{attribute 'linkalways'} 
{attribute 'no_explicit_call' := 'This FB is a CLASS and must be accessed using methods or properties'}
{attribute 'enable_dynamic_creation'}
{attribute 'hide_all_locals'}
FUNCTION_BLOCK PUBLIC FINAL List EXTENDS Disposable IMPLEMENTS I_List
VAR
	memoryManager : FB_DynMem_Manager2;
	buffer : FB_DynMem_Buffer(ipMemMan := memoryManager);
	pArrayOfListNodes : POINTER TO I_ListNode;
	arrayCapacity : DINT;
	itemCount : DINT;
	eventEmitter : EventEmitter;
END_VAR

METHOD PUBLIC AddItem
VAR_INPUT
	Item : ANY;
END_VAR
VAR
	node : I_ListNode;
END_VAR
node := CreateNewNode(Item);
IF AddNodeLast(node) THEN
	EmitChangedEvent();
END_IF
END_METHOD

METHOD PRIVATE AddNodeAt : BOOL
VAR_INPUT
	Index : DINT;
	Node : I_ListNode;
END_VAR
VAR
	i : DINT;
END_VAR
IF Index = itemCount THEN
	IF AddNodeLast(Node) THEN
		AddNodeAt := TRUE;
	END_IF
	RETURN;
END_IF

IF Index > itemCount - 1 THEN
	RETURN;
END_IF

IF itemCount + 1 > arrayCapacity THEN
	IF NOT Grow() THEN
		RETURN;
	END_IF
END_IF

IF IsBufferPointerValid THEN
	//Move all excisting nodes up
	FOR i := itemCount - 1 TO Index BY -1 DO
		pArrayOfListNodes[i + 1] := pArrayOfListNodes[i];
		pArrayOfListNodes[i] := 0;
	END_FOR
	
	pArrayOfListNodes[Index] := Node;
	itemCount := itemCount + 1;
	
	AddNodeAt := TRUE;
END_IF
END_METHOD

METHOD PRIVATE AddNodeLast : BOOL
VAR_INPUT
	Node : I_ListNode;
END_VAR
IF itemCount = arrayCapacity THEN
    IF NOT Grow() THEN
		RETURN;
	END_IF
END_IF

IF IsBufferPointerValid THEN
	pArrayOfListNodes[itemCount] := Node;
	itemCount := itemCount + 1;
	
	AddNodeLast := TRUE;
END_IF
END_METHOD

PROPERTY PUBLIC Capacity : DINT
GET
Capacity := arrayCapacity;
END_GET
END_PROPERTY

METHOD Clear
VAR_INPUT
END_VAR
IF IsEmpty THEN
	RETURN;
END_IF

RemoveAllNodes();
EmitChangedEvent();
END_METHOD

METHOD Contains : BOOL
VAR_INPUT
	Item : ANY;
END_VAR
IF IsEmpty THEN
	RETURN;
END_IF

Contains := GetIndexOf(Item) > -1;
END_METHOD

PROPERTY PUBLIC Count : DINT
GET
Count := itemCount;
END_GET
END_PROPERTY

METHOD PRIVATE CreateNewNode : I_ListNode
VAR_INPUT
	Value : ANY;
END_VAR
VAR
	pNode : POINTER TO ListNode;
END_VAR
pNode := __NEW(ListNode(Source := Value));
CreateNewNode := pNode^;
END_METHOD

METHOD PRIVATE EmitChangedEvent
VAR
	pCollectionChangedEvent : POINTER TO CollectionChangedEvent;
END_VAR
pCollectionChangedEvent := __NEW(CollectionChangedEvent(Target := THIS^));
eventEmitter.Emit('OnChanged', pCollectionChangedEvent^);
pCollectionChangedEvent^.Dispose();
END_METHOD

METHOD PRIVATE EmitDisposedEvent
VAR
	pCollectionDisposedEvent : POINTER TO CollectionDisposedEvent;
END_VAR
pCollectionDisposedEvent := __NEW(CollectionDisposedEvent(Target := THIS^));
eventEmitter.Emit('OnDisposed', pCollectionDisposedEvent^);
pCollectionDisposedEvent^.Dispose();
END_METHOD

METHOD FB_exit : BOOL
VAR_INPUT
	bInCopyCode : BOOL; // if TRUE, the exit method is called for exiting an instance that is copied afterwards (online change).
END_VAR
VAR
END_VAR
IF bInCopyCode THEN
    RETURN;
END_IF

Clear();
buffer.DeleteBuffer();
EmitDisposedEvent();
END_METHOD

METHOD GetEnumerator : I_ForwardEnumerator
VAR
	pEnumerator : POINTER TO ListForwardEnumerator;
END_VAR
pEnumerator := __NEW(ListForwardEnumerator(Parent := THIS^));
GetEnumerator := pEnumerator^;
END_METHOD

METHOD PUBLIC GetIndexOf : DINT
VAR_INPUT
	Item : ANY;
END_VAR
VAR
	node : I_ListNode;
	i : DINT;
END_VAR
GetIndexOf := -1;

IF IsEmpty THEN
	RETURN;
END_IF

FOR i := 0 TO itemCount - 1 DO
	node := THIS^.Item(i);
	
	IF node.Equals(Item) THEN
		GetIndexOf := i;
		RETURN;
	END_IF
END_FOR
END_METHOD

METHOD PRIVATE Grow : BOOL
VAR
	node : I_ListNode;
END_VAR
VAR CONSTANT
	INITIAL_CAPACITY : DINT := 4;
END_VAR
IF arrayCapacity = 0 THEN
	arrayCapacity := INITIAL_CAPACITY;
ELSE
	arrayCapacity := arrayCapacity * 2;
END_IF

IF buffer.bAvailable THEN
	IF NOT buffer.Resize(nSize := DINT_TO_UDINT(arrayCapacity) * SIZEOF(node), bPreserve := TRUE, bReset := FALSE) THEN
		RETURN;
	END_IF
ELSE
	IF NOT buffer.CreateBuffer(nSize := DINT_TO_UDINT(arrayCapacity) * SIZEOF(node), bReset := TRUE) THEN
		RETURN;
	END_IF
END_IF

IF buffer.bAvailable THEN
	pArrayOfListNodes := buffer.pBuffer;
	
	IF IsBufferPointerValid THEN
		Grow := TRUE;
	END_IF
END_IF
END_METHOD

PROPERTY PRIVATE IsBufferPointerValid : BOOL
GET
IsBufferPointerValid := pArrayOfListNodes <> 0;
END_GET
END_PROPERTY

PROPERTY IsEmpty : BOOL
GET
IsEmpty := itemCount = 0;
END_GET
END_PROPERTY

METHOD PRIVATE IsNotValidIndex : BOOL
VAR_INPUT
	Index : DINT;
END_VAR
IsNotValidIndex := NOT IsValidIndex(Index);
END_METHOD

METHOD PRIVATE IsValidIndex : BOOL
VAR_INPUT
	Index : DINT;
END_VAR
IF Index < 0 THEN
	RETURN;
END_IF

IF Index >= itemCount THEN
	RETURN;
END_IF

IsValidIndex := TRUE;
END_METHOD

METHOD PRIVATE Item : I_ListNode
VAR_INPUT
	Index : DINT;
END_VAR
IF IsNotValidIndex(Index) THEN
	RETURN;
END_IF

IF IsBufferPointerValid THEN
	Item := pArrayOfListNodes[Index];
END_IF
END_METHOD

METHOD PUBLIC OffEvent
VAR_INPUT
	EventName : T_MaxString;
	EventHandler : I_EventHandler;
END_VAR
eventEmitter.OffEvent(EventName, EventHandler);
END_METHOD

METHOD PUBLIC OnceEvent
VAR_INPUT
	EventName : T_MaxString;
	EventHandler : I_EventHandler;
END_VAR
eventEmitter.OnceEvent(EventName, EventHandler);
END_METHOD

METHOD PUBLIC OnEvent
VAR_INPUT
	EventName : T_MaxString;
	EventHandler : I_EventHandler;
END_VAR
eventEmitter.OnEvent(EventName, EventHandler);
END_METHOD

METHOD PRIVATE RemoveAllNodes
VAR
	i : DINT;
END_VAR
FOR i := 0 TO itemCount - 1 DO
	IF pArrayOfListNodes[i] <> 0 THEN
		pArrayOfListNodes[i].Dispose();
	END_IF
END_FOR

itemCount := 0;
END_METHOD

METHOD PUBLIC TrimExcess
VAR
	node : I_ListNode;
END_VAR
IF arrayCapacity = 0 THEN
	RETURN;
END_IF

IF arrayCapacity = itemCount THEN
	RETURN;
END_IF

arrayCapacity := itemCount;
IF buffer.Resize(nSize := DINT_TO_UDINT(arrayCapacity) * SIZEOF(node), bPreserve := TRUE, bReset := FALSE) THEN
	pArrayOfListNodes := buffer.pBuffer;
ELSE
	pArrayOfListNodes := 0;
END_IF
END_METHOD

METHOD PUBLIC TryCopyTo : BOOL
VAR_INPUT
	Destination	: ANY;
END_VAR
TryCopyTo := TryCopyToLocation(Destination.pValue, DINT_TO_UDINT(Destination.diSize));
END_METHOD

METHOD PUBLIC TryCopyToLocation : BOOL
VAR_INPUT
	DestinationAddress : PVOID;
	DestinationSize : UDINT;
END_VAR
VAR
	i : DINT;
	requiredSize : UDINT;
	current : I_ListNode;
	pCurrent : PVOID;
END_VAR
IF IsEmpty THEN
    RETURN;
END_IF

//Compute required size
FOR i := 0 TO Count - 1 DO
    current := Item(i);
    requiredSize := requiredSize + current.DataSize;
END_FOR

//If destination size is to small abort
IF DestinationSize < requiredSize THEN
    RETURN;
END_IF

pCurrent := DestinationAddress;

FOR i := 0 TO Count - 1 DO
    current := Item(i);
    current.TryGetTo(pCurrent, current.DataSize);
    pCurrent := pCurrent + current.DataSize;
END_FOR
END_METHOD

METHOD PUBLIC TryGetByIndex : BOOL
VAR_INPUT
	Index : DINT;
	Destination : ANY;
END_VAR
VAR
	node : I_ListNode;
END_VAR
node := Item(Index);

IF node = 0 THEN
	RETURN;
END_IF

TryGetByIndex := node.TryGet(Destination);
END_METHOD

METHOD PUBLIC TryGetToByIndex : BOOL
VAR_INPUT
	Index : DINT;
	DestinationAddress : PVOID;
	DestinationSize : UDINT;
END_VAR
VAR
	node : I_ListNode;
END_VAR
node := Item(Index);

IF node = 0 THEN
	RETURN;
END_IF

TryGetToByIndex := node.TryGetTo(DestinationAddress, DestinationSize);
END_METHOD

METHOD TryInsert : BOOL
VAR_INPUT
	Index : DINT;
	Item : ANY;
END_VAR
VAR
	node : I_ListNode;
END_VAR
IF IsNotValidIndex(Index) THEN
	RETURN;
END_IF

node := CreateNewNode(Item);
IF AddNodeAt(Index, node) THEN
	EmitChangedEvent();
	TryInsert := TRUE;
END_IF
END_METHOD

METHOD PUBLIC TryRemoveAt : BOOL;
VAR_INPUT
	Index : DINT;
END_VAR
VAR
	i : DINT;
	node : I_ListNode;
END_VAR
IF IsNotValidIndex(Index) THEN
	RETURN;
END_IF

IF IsBufferPointerValid THEN
	node := Item(Index);
	node.Dispose();
	
	FOR i := Index + 1 TO itemCount - 1 DO
		pArrayOfListNodes[i - 1] := pArrayOfListNodes[i];
		pArrayOfListNodes[i] := 0;
	END_FOR
	
	itemCount := itemCount - 1;
	EmitChangedEvent();
	TryRemoveAt := TRUE;
END_IF
END_METHOD

METHOD TryRemoveItem : BOOL
VAR_INPUT
    Item : ANY;
END_VAR
VAR
    index : DINT;
END_VAR
index := GetIndexOf(Item);

IF index = -1 THEN
	RETURN;
END_IF

TryRemoveItem := TryRemoveAt(index);
END_METHOD

END_FUNCTION_BLOCK

(* stored: Version 1.1.0.1, ProductVersion 3.1.4026.6
   POU List: Id {9220d5a8-4969-08a4-1724-7633ca12bf29}, SpecialFunc None
   Folder Destructor: Id {8fdd593d-4b5b-0cba-142b-2136390a5ba1}
   Folder Private: Id {f8e6fb94-8042-49e9-832d-ab6b0922fdf1}
   Method AddItem: Id {4338eac4-cb94-0e48-0359-63eec208e760}
   Method AddNodeAt: Id {434fcbfc-1b21-406c-bc70-53644c6aca95}
   Method AddNodeLast: Id {0fd32a56-42dd-46f2-9f6e-72084c72716b}
   Property Capacity: Id {627ddc89-13f9-42d2-99f0-470fa6c85ab9}
   Get Get: Id {e1b9172c-d486-48b5-afdf-e3673af87d0e}
   Method Clear: Id {6a51ab3d-5d81-406b-91df-b56045948387}
   Method Contains: Id {8d070616-89e9-48db-8902-c17e7098b90d}
   Property Count: Id {18af26e5-6368-08f4-3269-b1e13029edb8}
   Get Get: Id {84d29658-765a-06de-2dbc-7bd104ca837e}
   Method CreateNewNode: Id {669eec89-9d9f-4b2d-8f7d-4af8a72f842c}
   Method EmitChangedEvent: Id {ca89fe9e-ace0-4c15-b1dc-fef757879f08}
   Method EmitDisposedEvent: Id {880ec866-3d07-4171-8716-ab03bbbd8f1f}
   Method FB_exit: Id {a189a9f3-674e-0a1c-24b3-a20087e08971}
   Method GetEnumerator: Id {fea1fcad-e669-422d-9653-a618518cd1c8}
   Method GetIndexOf: Id {11432220-b6bf-4ad5-94bd-7b00101eef0a}
   Method Grow: Id {aa524b81-d1fc-4fc5-8e9b-5c5798157c90}
   Property IsBufferPointerValid: Id {050ffdb2-bc7f-4534-a751-06f0e5aa65c5}
   Get Get: Id {343b014d-2e57-4916-aada-74911f7348c5}
   Property IsEmpty: Id {4ad381b9-db6e-4adb-9e4a-12902170c312}
   Get Get: Id {a9e217e4-6ded-4f1a-9d8d-aadaebe0bcf4}
   Method IsNotValidIndex: Id {6b2f0604-0d45-4dec-b1e4-88140675f855}
   Method IsValidIndex: Id {509f1c3a-d218-4854-ab0e-56d9f99586ec}
   Method Item: Id {5f4268ee-abf7-400e-939d-8a03550a5e63}
   Method OffEvent: Id {6d43365d-a3f5-40bf-b0a0-cad17bdad2f3}
   Method OnceEvent: Id {9955174c-27ac-48f9-a497-6248067945ea}
   Method OnEvent: Id {c2d02837-c38b-41f8-8beb-7c48b9d725f4}
   Method RemoveAllNodes: Id {1924a692-4a0d-400c-b4f6-02313ee91984}
   Method TrimExcess: Id {6de9ea7b-ef6a-4934-859f-de170f7ffff9}
   Method TryCopyTo: Id {08647dfb-c5bf-4481-b560-e5f349a8a87f}
   Method TryCopyToLocation: Id {2460292a-feaa-4f20-a5c3-9f55d0dc2c6c}
   Method TryGetByIndex: Id {58aae7f1-11d1-4b34-9d25-48c86c9e3f03}
   Method TryGetToByIndex: Id {300cb5be-24cb-4729-a1a8-f89043705dd7}
   Method TryInsert: Id {4a28931b-7145-4a14-a1cc-726d2ed98557}
   Method TryRemoveAt: Id {5fddda2d-2bc3-08a7-1fc5-3303b29b003f}
   Method TryRemoveItem: Id {405b8587-bb35-4a7f-9adc-3766cc05ff19} *)
